	FUNCTION_BLOCK FB 397
	TITLE =G297M FAN KILN 2
	//COPYRIGHT:    (C) 2009  BUHLER AG, CH-9240 UZWIL, SWITZERLAND
	//
	//PRODUCT:      WinCoS_BIW01_09
	//
	//TITLE:        FAN KILN 2
	//                Machine group control
	//                Maschinengruppensteuerung
	//
	//--------------------------------------------------------------------------------
	//
	//IDENT:        AUTHOR:             DEPT:                              DATE:
	//
	//P01_FB397.1.0 K.Renz              CSB41                              20.Mai.2010
	//             1st Release
	//
	//--------------------------------------------------------------------------------
	//
	//PURPOSE:
	//
	//MANUAL :
	//
	//RESTRICTIONS:
	//
	//--------------------------------------------------------------------------------
	AUTHOR  : KR
	FAMILY  : USW
	VERSION : 9.9


	VAR
	  Gr       : FB10;	//Standard interface to group
	  InOutValue1    : DINT; //Data for user
	  InOutValue2    : DINT; //Data for user
	  OutWayConflict : BOOL;	//Data for user
	  OutSelectionOk : BOOL;	//Data for user
	  CmdNewValue : BOOL;	//Data for user
	  CmdNewJob   : BOOL;	//Data for user
	  OutCodeOK   : BOOL;	//Data for user
	  InEndOfJob  : BOOL ;	//Data for user
	  staWayOk      : BOOL ;	//Data for user
	  EdgeStartRelease : BOOL ;	//Data for user
	  USW8  : BOOL;	//Data for user
	  USW9 : BOOL;	//Data for user
	  USW10: BOOL;	//Data for user
	  USW11: BOOL;	//Data for user
	  USW12: BOOL;	//Data for user
	  USW13: BOOL;	//Data for user
	  USW14: BOOL;	//Data for user
	  USW15: BOOL;	//Data for user
	     #A_3225_KCU04AI1 : FB19;   // AnaInp
	     #A_3225_KCU04AI2 : FB19;   // AnaInp
	     #A_3225_BTE05 : FB19;   // AnaInp
	     #A_3225_BTE06 : FB19;   // AnaInp
	     #A_3225_TSC01 : FB14;   // DigInpCont
	     #A_3225_MXZ01MA : FB1032;   // Motor+6DI
	     #A_3225_TSC01_AC : FB19;   // AnaInp
	     #A_3225_TSC01_AF : FB19;   // AnaInp
	     #A_3225_TSC01_AP : FB19;   // AnaInp
	     #A_3225_TSC01_AT : FB19;   // AnaInp
	     #A_3225_TSC01_COM : FB1812;   // FU_Siemens
	     #A_3226_KCU04AI1 : FB19;   // AnaInp
	     #A_3226_KCU04AI2 : FB19;   // AnaInp
	     #A_3226_BTE05 : FB19;   // AnaInp
	     #A_3226_BTE06 : FB19;   // AnaInp
	     #A_3226_MXZ01MA : FB1033;   // Motor+6DI
	     #A_3226_TSC01_AC : FB19;   // AnaInp
	     #A_3226_TSC01_AF : FB19;   // AnaInp
	     #A_3226_TSC01_AP : FB19;   // AnaInp
	     #A_3226_TSC01_AT : FB19;   // AnaInp
	     #A_3226_TSC01_COM : FB1812;   // FU_Siemens
	     #A_3226_TSC01 : FB14;   // DigInpCont
	     #A_3225_MXZ02MA : FB1066;   // Motor+6DI
	     #A_3226_MXZ02MA : FB1067;   // Motor+6DI
	END_VAR
	VAR_TEMP
	   tmpEnable		: BOOL;
	   tmpFlag  		: BOOL;
	   tmpCmdNext		: BOOL;
	   tmpLocal  		: BOOL;
	   tmpAspOk  		: BOOL;
	   tmpHWStop 		: BOOL;
	   tmpInstanzDBNo       : INT ;
	END_VAR
	BEGIN
	NETWORK
	TITLE =
	NETWORK
	TITLE =Read command from group control
	//Parameter
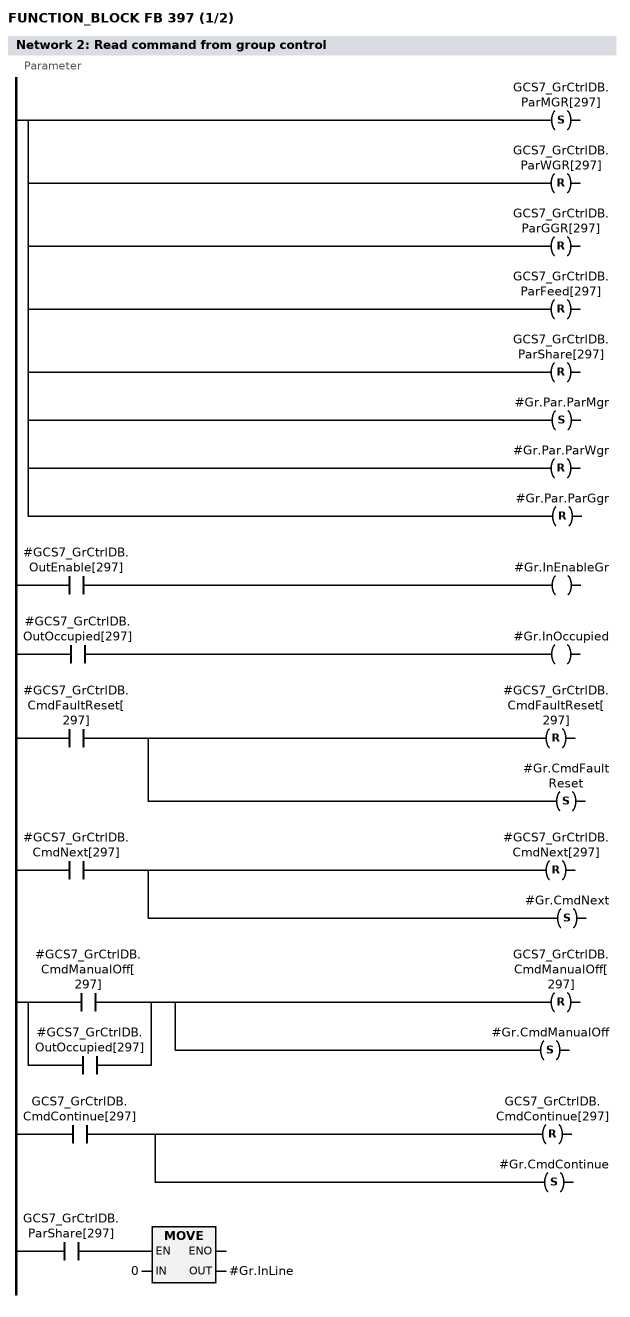
	      SET;
	      S   GCS7_GrCtrlDB.ParMGR[297];
	      R   GCS7_GrCtrlDB.ParWGR[297];
	      R   GCS7_GrCtrlDB.ParGGR[297];
	      R   GCS7_GrCtrlDB.ParFeed[297];
	      R   GCS7_GrCtrlDB.ParShare[297];
	      S   #Gr.Par.ParMgr;
	      R   #Gr.Par.ParWgr;
	      R   #Gr.Par.ParGgr;
	//Command
	      U   #GCS7_GrCtrlDB.OutEnable[297];
	      =   #Gr.InEnableGr;
	      U   #GCS7_GrCtrlDB.OutOccupied[297];
	      =   #Gr.InOccupied;
	      U   #GCS7_GrCtrlDB.CmdFaultReset[297];
	      R   #GCS7_GrCtrlDB.CmdFaultReset[297];
	      S   #Gr.CmdFaultReset;
	      U  #GCS7_GrCtrlDB.CmdNext[297];
	      R   #GCS7_GrCtrlDB.CmdNext[297];
	      S   #Gr.CmdNext;
	      U   #GCS7_GrCtrlDB.CmdManualOff[297];
	      O   #GCS7_GrCtrlDB.OutOccupied[297];
	      R   GCS7_GrCtrlDB.CmdManualOff[297];
	      S   #Gr.CmdManualOff;
	      U  GCS7_GrCtrlDB.CmdContinue[297];
	      R   GCS7_GrCtrlDB.CmdContinue[297];
	      S   #Gr.CmdContinue;
	//Init Line Number
	      U   GCS7_GrCtrlDB.ParShare[297];
	      SPBN WE00;
	      L     0;
	      T     #Gr.InLine;
	WE00: NOP   0;
	NETWORK
	TITLE =Call Methode Control
	// 1. Handle Interface PCControl
	// 2. Prepare mode --> ModePassive,ModeActive,ModeIdling
	// 3. Reset global flags of the group
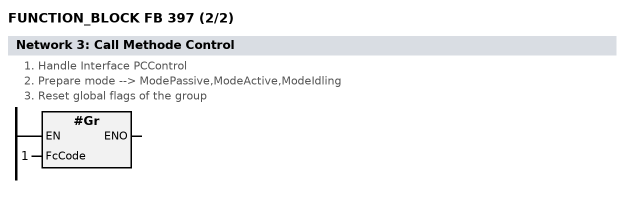
	      CALL #Gr (
	           FcCode                   := 1);
	NETWORK
	TITLE =Restart Idling Time
		L  #Gr.Par.ParIdling;
		L  2;
		>=I;
		SPB IdTm;
		T  #Gr.Par.ParIdling;
	IdTm:   NOP 0;
	      CLR;
	      S    #Gr.CmdRestartIdling;
	NETWORK
	TITLE =Prepare global flags
	NETWORK
	TITLE =Set Pattern (Target position)
	NETWORK
	TITLE =Interlocking WayOk
	//
	NETWORK
	TITLE =Interlocking Autostart
		CLR;
		R   #Gr.OutAutostart;
	NETWORK
	TITLE =Interlocking Enable
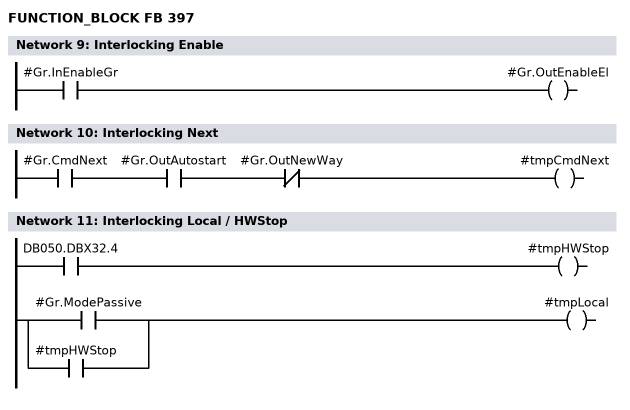
	      U     #Gr.InEnableGr;
	      =     #Gr.OutEnableEl;

	NETWORK
	TITLE =Interlocking Next
	      U     #Gr.CmdNext;
	      U     #Gr.OutAutostart;
	      UN    #Gr.OutNewWay;
	      =    #tmpCmdNext;

	NETWORK
	TITLE =Interlocking Local / HWStop
	      U    DB050.DBX32.4;
	      =    #tmpHWStop;

	      U    #Gr.ModePassive;
	      O    #tmpHWStop;
	      =    #tmpLocal;

	NETWORK
	TITLE =Interlocking Start Warning
	      NOP 0;
	//- Restart after fault --
	      U     #Gr.CmdFaultReset;
	      U     #Gr.VarFault;
	      S       "SYS_StartWarningDB".Area[11].CmdResetStartWarning;
	//- Run Timer --
	      AUF "G297M";
	      CALL  FB100 , DB100(
	       InModeHigher :=FALSE,
	       InArea     :=11,
	       InEnable   :=#Gr.OutEnableEl,
	       InLocal    :=#tmpLocal,
	       InStarted  :=#Gr.VarStarted,
	       InCmdNext  :=#tmpCmdNext,
	       OutCmdNext :=#tmpCmdNext,
	       OutStartwarning:=#Gr.VarStartWarning);
	//- Store Startwarning done  --
	//- Reset Autostart --
	      U     "SYS_StartWarningDB".TmpArea.OutStartReleaseRunningL;
	      FN    #EdgeStartRelease;
	      U     #Gr.VarFault;
	      R     #Gr.OutAutostart;
	NETWORK
	TITLE ==A-3225-KCU04AI1 : VIBRATION MONITOR FAN 1 CHANNEL 1
	NOP 0;
	//-InLocal---
	      U     #tmpLocal;
	      =     #A_3225_KCU04AI1.InLocal;
	//
	//-Monitoring---
	      CLR;
	      =     #A_3225_KCU04AI1.InMonLL;
	      CLR;
	      =     #A_3225_KCU04AI1.InMonL;
	      CLR;
	      =     #A_3225_KCU04AI1.InMonMid;
	      CLR;
	      =     #A_3225_KCU04AI1.InMonH;
	      SET;
	      =     #A_3225_KCU04AI1.InMonHH;
	//
	//-Read inputs---
	      L     PEW1054;
	      T     #A_3225_KCU04AI1.InpValue;
	      U   DB050.DBX32.4;
	      =     #A_3225_KCU04AI1.InHWStop;
	       U     PLC_DPInfo.Master[1].SlavesError[102];
	       =       #A_3225_KCU04AI1.InDPFault;
	//
	//-Set Parameters---
	//
	//-Call object control---
	      CALL  #A_3225_KCU04AI1;
	//
	//-Write outputs---
	NETWORK
	TITLE ==A-3225-KCU04AI2 : VIBRATION MONITOR FAN 1 CHANNEL 2
	NOP 0;
	//-InLocal---
	      U     #tmpLocal;
	      =     #A_3225_KCU04AI2.InLocal;
	//
	//-Monitoring---
	      CLR;
	      =     #A_3225_KCU04AI2.InMonLL;
	      CLR;
	      =     #A_3225_KCU04AI2.InMonL;
	      CLR;
	      =     #A_3225_KCU04AI2.InMonMid;
	      CLR;
	      =     #A_3225_KCU04AI2.InMonH;
	      SET;
	      =     #A_3225_KCU04AI2.InMonHH;
	//
	//-Read inputs---
	      L     PEW1052;
	      T     #A_3225_KCU04AI2.InpValue;
	      U   DB050.DBX32.4;
	      =     #A_3225_KCU04AI2.InHWStop;
	       U     PLC_DPInfo.Master[1].SlavesError[102];
	       =       #A_3225_KCU04AI2.InDPFault;
	//
	//-Set Parameters---
	//
	//-Call object control---
	      CALL  #A_3225_KCU04AI2;
	//
	//-Write outputs---
	NETWORK
	TITLE ==A-3225-BTE05 : TEMPERATURE BEARING TEMPERATUR SENSOR
	NOP 0;
	//-InLocal---
	      U     #tmpLocal;
	      =     #A_3225_BTE05.InLocal;
	//
	//-Monitoring---
	      CLR;
	      =     #A_3225_BTE05.InMonLL;
	      CLR;
	      =     #A_3225_BTE05.InMonL;
	      CLR;
	      =     #A_3225_BTE05.InMonMid;
	      CLR;
	      =     #A_3225_BTE05.InMonH;
	      SET;
	      =     #A_3225_BTE05.InMonHH;
	//
	//-Read inputs---
	      L     PEW1028;
	      T     #A_3225_BTE05.InpValue;
	      U   DB050.DBX32.4;
	      =     #A_3225_BTE05.InHWStop;
	       U     PLC_DPInfo.Master[1].SlavesError[102];
	       =       #A_3225_BTE05.InDPFault;
	//
	//-Set Parameters---
	//
	//-Call object control---
	      CALL  #A_3225_BTE05;
	//
	//-Write outputs---
	NETWORK
	TITLE ==A-3225-BTE06 : TEMPERATURE BEARING TEMPERATUR SENSOR
	NOP 0;
	//-InLocal---
	      U     #tmpLocal;
	      =     #A_3225_BTE06.InLocal;
	//
	//-Monitoring---
	      CLR;
	      =     #A_3225_BTE06.InMonLL;
	      CLR;
	      =     #A_3225_BTE06.InMonL;
	      CLR;
	      =     #A_3225_BTE06.InMonMid;
	      CLR;
	      =     #A_3225_BTE06.InMonH;
	      SET;
	      =     #A_3225_BTE06.InMonHH;
	//
	//-Read inputs---
	      L     PEW1030;
	      T     #A_3225_BTE06.InpValue;
	      U   DB050.DBX32.4;
	      =     #A_3225_BTE06.InHWStop;
	       U     PLC_DPInfo.Master[1].SlavesError[102];
	       =       #A_3225_BTE06.InDPFault;
	//
	//-Set Parameters---
	//
	//-Call object control---
	      CALL  #A_3225_BTE06;
	//
	//-Write outputs---
	NETWORK
	TITLE ==A-3225-MXZ02MA : GETRIEBEÖLPUMPE FAN 1
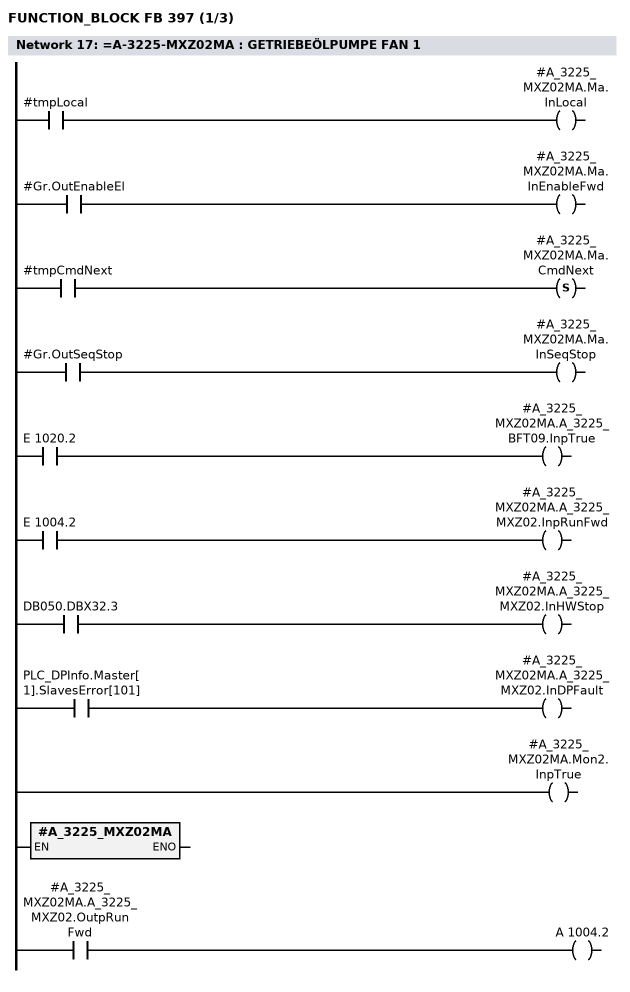
	NOP 0;
	//-InLocal---
	      U     #tmpLocal;
	      =     #A_3225_MXZ02MA.Ma.InLocal;
	//
	//-Interlocking---

	      U     #Gr.OutEnableEl;
	      =     #A_3225_MXZ02MA.Ma.InEnableFwd;
	//
	      U    #tmpCmdNext;
	      S     #A_3225_MXZ02MA.Ma.CmdNext;
	//
	      U     #Gr.OutSeqStop;
	      =     #A_3225_MXZ02MA.Ma.InSeqStop;
	//
	//=Values and commands of elements===
	//-=A-3225-BFT09---
	//      CLR
	//      S     #A_3225_MXZ02MA.A_3225_BFT09.CmdRunTimeOutTime
	//
	//-Read inputs of elements---
	      U     E 1020.2;
	      =     #A_3225_MXZ02MA.A_3225_BFT09.InpTrue;
	      U     E 1004.2;
	      =     #A_3225_MXZ02MA.A_3225_MXZ02.InpRunFwd;
	      U   DB050.DBX32.3;
	      =     #A_3225_MXZ02MA.A_3225_MXZ02.InHWStop;
	       U     PLC_DPInfo.Master[1].SlavesError[101];
	       =       #A_3225_MXZ02MA.A_3225_MXZ02.InDPFault;
	      SET;
	      =     #A_3225_MXZ02MA.Mon2.InpTrue;
	//
	//-Set Parameters---
	//
	//-Call object control---
	      CALL  #A_3225_MXZ02MA;
	//
	//-Write outputs---
	      U     #A_3225_MXZ02MA.A_3225_MXZ02.OutpRunFwd;
	      =     A 1004.2;
	NETWORK
	TITLE ==A-3225-MXZ01MA : FAN 1
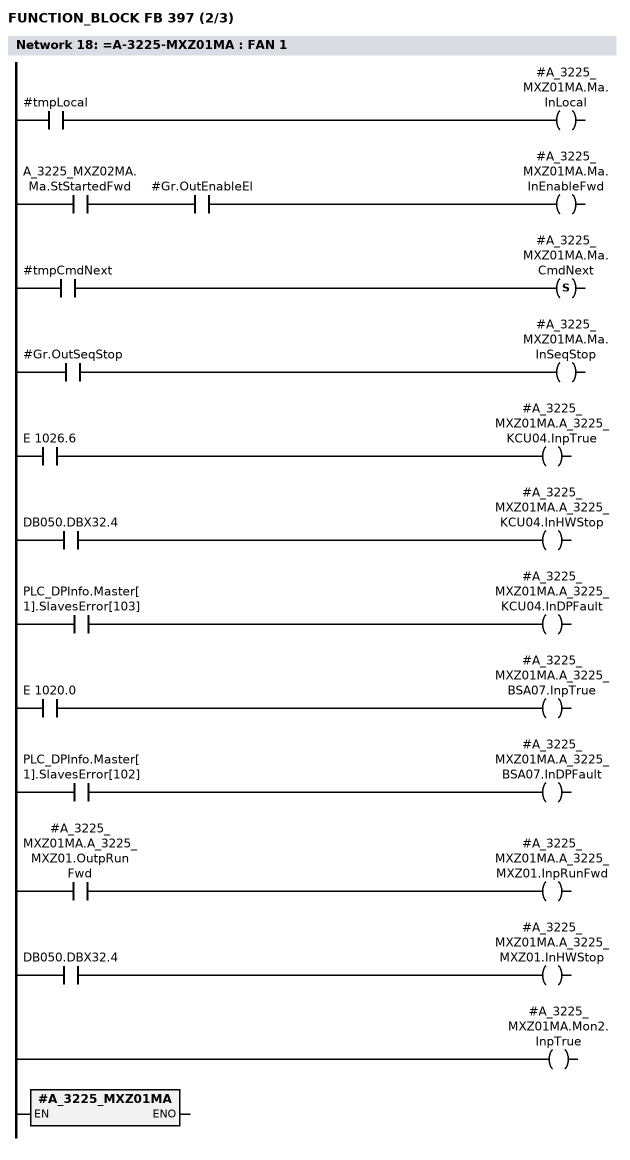
	NOP 0;
	//-InLocal---
	      U     #tmpLocal;
	      =     #A_3225_MXZ01MA.Ma.InLocal;
	//
	//-Interlocking---
	      U A_3225_MXZ02MA.Ma.StStartedFwd;
	      U     #Gr.OutEnableEl;
	      =     #A_3225_MXZ01MA.Ma.InEnableFwd;
	//
	      U    #tmpCmdNext;
	      S     #A_3225_MXZ01MA.Ma.CmdNext;
	//
	      U     #Gr.OutSeqStop;
	      =     #A_3225_MXZ01MA.Ma.InSeqStop;
	//
	//=Values and commands of elements===
	//-=A-3225-KCU04---
	//      CLR
	//      S     #A_3225_MXZ01MA.A_3225_KCU04.CmdRunTimeOutTime
	//-=A-3225-BSA07---
	//      CLR
	//      S     #A_3225_MXZ01MA.A_3225_BSA07.CmdRunTimeOutTime
	//
	//-Read inputs of elements---
	      U     E 1026.6;
	      =     #A_3225_MXZ01MA.A_3225_KCU04.InpTrue;
	      U   DB050.DBX32.4;
	      =     #A_3225_MXZ01MA.A_3225_KCU04.InHWStop;
	       U     PLC_DPInfo.Master[1].SlavesError[103];
	       =       #A_3225_MXZ01MA.A_3225_KCU04.InDPFault;
	      U     E 1020.0;
	      =     #A_3225_MXZ01MA.A_3225_BSA07.InpTrue;
	       U     PLC_DPInfo.Master[1].SlavesError[102];
	       =       #A_3225_MXZ01MA.A_3225_BSA07.InDPFault;
	      U     #A_3225_MXZ01MA.A_3225_MXZ01.OutpRunFwd;
	      =     #A_3225_MXZ01MA.A_3225_MXZ01.InpRunFwd;
	      U   DB050.DBX32.4;
	      =     #A_3225_MXZ01MA.A_3225_MXZ01.InHWStop;
	      SET;
	      =     #A_3225_MXZ01MA.Mon2.InpTrue;
	//
	//-Set Parameters---
	//
	//-Call object control---
	      CALL  #A_3225_MXZ01MA;
	//
	//-Write outputs---
	NETWORK
	TITLE ==A-3225-TSC01_COM : FAN 1 FU KOMMUNIKATION
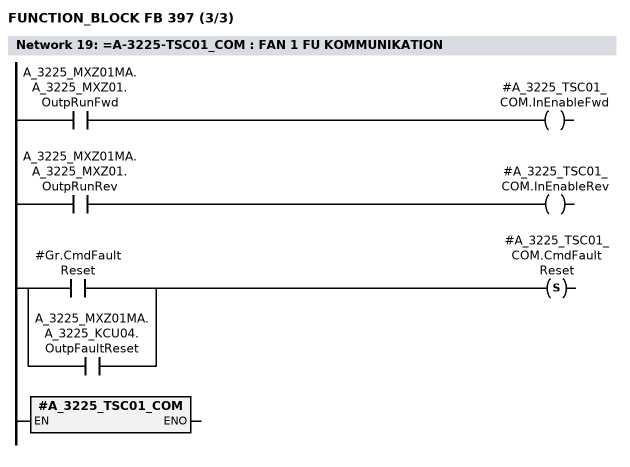
	NOP 0;
	     U   A_3225_MXZ01MA.A_3225_MXZ01.OutpRunFwd;
	      =     #A_3225_TSC01_COM.InEnableFwd;
	     U    A_3225_MXZ01MA.A_3225_MXZ01.OutpRunRev;
	      =     #A_3225_TSC01_COM.InEnableRev;
	     U     #Gr.CmdFaultReset;
	     O    A_3225_MXZ01MA.A_3225_KCU04.OutpFaultReset;
	      S     #A_3225_TSC01_COM.CmdFaultReset;
	//
	//
	//-Read inputs---
	//
	//-Set Parameters---
	//
	//-Call object control---
	      CALL  #A_3225_TSC01_COM;
	//
	//-Write outputs---
	NETWORK
	TITLE ==A-3225-TSC01_AC : ACT. CURRENT FAN 1 FU
	NOP 0;
	//-InLocal---
	      U     #tmpLocal;
	      =     #A_3225_TSC01_AC.InLocal;
	//
	//-Monitoring---
	      CLR;
	      =     #A_3225_TSC01_AC.InMonLL;
	      CLR;
	      =     #A_3225_TSC01_AC.InMonL;
	      CLR;
	      =     #A_3225_TSC01_AC.InMonMid;
	      CLR;
	      =     #A_3225_TSC01_AC.InMonH;
	      CLR;
	      =     #A_3225_TSC01_AC.InMonHH;
	//
	//-Read inputs---
	      L     A_3225_TSC01_COM.Output.SetpointValue01;
	      ITD;
	      DTR;
	      ABS;
	      RND;
	      T     #A_3225_TSC01_AC.InpValue;
	      U   DB050.DBX32.4;
	      =     #A_3225_TSC01_AC.InHWStop;
	//
	//-Set Parameters---
	//
	//-Call object control---
	      CALL  #A_3225_TSC01_AC;
	//
	//-Write outputs---
	NETWORK
	TITLE ==A-3225-TSC01_AF : ACT. FREQUENCY FAN 1 FU
	NOP 0;
	//-InLocal---
	      U     #tmpLocal;
	      =     #A_3225_TSC01_AF.InLocal;
	//
	//-Monitoring---
	      CLR;
	      =     #A_3225_TSC01_AF.InMonLL;
	      CLR;
	      =     #A_3225_TSC01_AF.InMonL;
	      CLR;
	      =     #A_3225_TSC01_AF.InMonMid;
	      CLR;
	      =     #A_3225_TSC01_AF.InMonH;
	      CLR;
	      =     #A_3225_TSC01_AF.InMonHH;
	//
	//-Read inputs---
	      L     A_3225_TSC01_COM.Output.SetpointValue01;
	      ITD;
	      DTR;
	      ABS;
	      RND;
	      T     #A_3225_TSC01_AF.InpValue;
	      U   DB050.DBX32.4;
	      =     #A_3225_TSC01_AF.InHWStop;
	//
	//-Set Parameters---
	//
	//-Call object control---
	      CALL  #A_3225_TSC01_AF;
	//
	//-Write outputs---
	NETWORK
	TITLE ==A-3225-TSC01_AP : ACT. POWER FAN 1 FU
	NOP 0;
	//-InLocal---
	      U     #tmpLocal;
	      =     #A_3225_TSC01_AP.InLocal;
	//
	//-Monitoring---
	      CLR;
	      =     #A_3225_TSC01_AP.InMonLL;
	      CLR;
	      =     #A_3225_TSC01_AP.InMonL;
	      CLR;
	      =     #A_3225_TSC01_AP.InMonMid;
	      CLR;
	      =     #A_3225_TSC01_AP.InMonH;
	      CLR;
	      =     #A_3225_TSC01_AP.InMonHH;
	//
	//-Read inputs---
	      L     A_3225_TSC01_COM.Output.SetpointValue01;
	      ITD;
	      DTR;
	      ABS;
	      RND;
	      T     #A_3225_TSC01_AP.InpValue;
	      U   DB050.DBX32.4;
	      =     #A_3225_TSC01_AP.InHWStop;
	//
	//-Set Parameters---
	//
	//-Call object control---
	      CALL  #A_3225_TSC01_AP;
	//
	//-Write outputs---
	NETWORK
	TITLE ==A-3225-TSC01_AT : ACT. TORQUE FAN 1 FU
	NOP 0;
	//-InLocal---
	      U     #tmpLocal;
	      =     #A_3225_TSC01_AT.InLocal;
	//
	//-Monitoring---
	      CLR;
	      =     #A_3225_TSC01_AT.InMonLL;
	      CLR;
	      =     #A_3225_TSC01_AT.InMonL;
	      CLR;
	      =     #A_3225_TSC01_AT.InMonMid;
	      CLR;
	      =     #A_3225_TSC01_AT.InMonH;
	      CLR;
	      =     #A_3225_TSC01_AT.InMonHH;
	//
	//-Read inputs---
	      L     A_3225_TSC01_COM.Output.SetpointValue01;
	      ITD;
	      DTR;
	      ABS;
	      RND;
	      T     #A_3225_TSC01_AT.InpValue;
	      U   DB050.DBX32.4;
	      =     #A_3225_TSC01_AT.InHWStop;
	//
	//-Set Parameters---
	//
	//-Call object control---
	      CALL  #A_3225_TSC01_AT;
	//
	//-Write outputs---
	NETWORK
	TITLE ==A-3226-KCU04AI1 : VIBRATION MONITOR FAN 2 CHANNEL 1
	NOP 0;
	//-InLocal---
	      U     #tmpLocal;
	      =     #A_3226_KCU04AI1.InLocal;
	//
	//-Monitoring---
	      CLR;
	      =     #A_3226_KCU04AI1.InMonLL;
	      CLR;
	      =     #A_3226_KCU04AI1.InMonL;
	      CLR;
	      =     #A_3226_KCU04AI1.InMonMid;
	      CLR;
	      =     #A_3226_KCU04AI1.InMonH;
	      SET;
	      =     #A_3226_KCU04AI1.InMonHH;
	//
	//-Read inputs---
	      L     PEW1058;
	      T     #A_3226_KCU04AI1.InpValue;
	      U   DB050.DBX32.4;
	      =     #A_3226_KCU04AI1.InHWStop;
	       U     PLC_DPInfo.Master[1].SlavesError[102];
	       =       #A_3226_KCU04AI1.InDPFault;
	//
	//-Set Parameters---
	//
	//-Call object control---
	      CALL  #A_3226_KCU04AI1;
	//
	//-Write outputs---
	NETWORK
	TITLE ==A-3226-KCU04AI2 : VIBRATION MONITOR FAN 2 CHANNEL 2
	NOP 0;
	//-InLocal---
	      U     #tmpLocal;
	      =     #A_3226_KCU04AI2.InLocal;
	//
	//-Monitoring---
	      CLR;
	      =     #A_3226_KCU04AI2.InMonLL;
	      CLR;
	      =     #A_3226_KCU04AI2.InMonL;
	      CLR;
	      =     #A_3226_KCU04AI2.InMonMid;
	      CLR;
	      =     #A_3226_KCU04AI2.InMonH;
	      SET;
	      =     #A_3226_KCU04AI2.InMonHH;
	//
	//-Read inputs---
	      L     PEW1056;
	      T     #A_3226_KCU04AI2.InpValue;
	      U   DB050.DBX32.4;
	      =     #A_3226_KCU04AI2.InHWStop;
	       U     PLC_DPInfo.Master[1].SlavesError[102];
	       =       #A_3226_KCU04AI2.InDPFault;
	//
	//-Set Parameters---
	//
	//-Call object control---
	      CALL  #A_3226_KCU04AI2;
	//
	//-Write outputs---
	NETWORK
	TITLE ==A-3226-BTE05 : TEMPERATURE BEARING TEMPERATUR SENSOR
	NOP 0;
	//-InLocal---
	      U     #tmpLocal;
	      =     #A_3226_BTE05.InLocal;
	//
	//-Monitoring---
	      CLR;
	      =     #A_3226_BTE05.InMonLL;
	      CLR;
	      =     #A_3226_BTE05.InMonL;
	      CLR;
	      =     #A_3226_BTE05.InMonMid;
	      CLR;
	      =     #A_3226_BTE05.InMonH;
	      SET;
	      =     #A_3226_BTE05.InMonHH;
	//
	//-Read inputs---
	      L     PEW1032;
	      T     #A_3226_BTE05.InpValue;
	      U   DB050.DBX32.4;
	      =     #A_3226_BTE05.InHWStop;
	       U     PLC_DPInfo.Master[1].SlavesError[102];
	       =       #A_3226_BTE05.InDPFault;
	//
	//-Set Parameters---
	//
	//-Call object control---
	      CALL  #A_3226_BTE05;
	//
	//-Write outputs---
	NETWORK
	TITLE ==A-3226-BTE06 : TEMPERATURE BEARING TEMPERATUR SENSOR
	NOP 0;
	//-InLocal---
	      U     #tmpLocal;
	      =     #A_3226_BTE06.InLocal;
	//
	//-Monitoring---
	      CLR;
	      =     #A_3226_BTE06.InMonLL;
	      CLR;
	      =     #A_3226_BTE06.InMonL;
	      CLR;
	      =     #A_3226_BTE06.InMonMid;
	      CLR;
	      =     #A_3226_BTE06.InMonH;
	      SET;
	      =     #A_3226_BTE06.InMonHH;
	//
	//-Read inputs---
	      L     PEW1034;
	      T     #A_3226_BTE06.InpValue;
	      U   DB050.DBX32.4;
	      =     #A_3226_BTE06.InHWStop;
	       U     PLC_DPInfo.Master[1].SlavesError[102];
	       =       #A_3226_BTE06.InDPFault;
	//
	//-Set Parameters---
	//
	//-Call object control---
	      CALL  #A_3226_BTE06;
	//
	//-Write outputs---
	NETWORK
	TITLE ==A-3226-MXZ02MA : GETRIEBEÖLPUMPE FAN 2
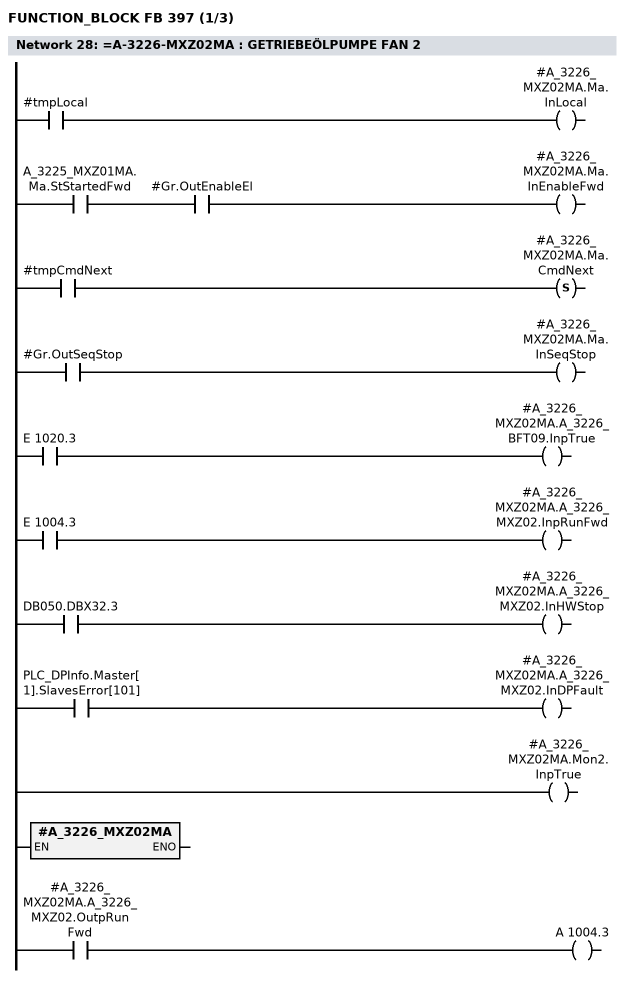
	NOP 0;
	//-InLocal---
	      U     #tmpLocal;
	      =     #A_3226_MXZ02MA.Ma.InLocal;
	//
	//-Interlocking---
	      U A_3225_MXZ01MA.Ma.StStartedFwd;
	      U     #Gr.OutEnableEl;
	      =     #A_3226_MXZ02MA.Ma.InEnableFwd;
	//
	      U    #tmpCmdNext;
	      S     #A_3226_MXZ02MA.Ma.CmdNext;
	//
	      U     #Gr.OutSeqStop;
	      =     #A_3226_MXZ02MA.Ma.InSeqStop;
	//
	//=Values and commands of elements===
	//-=A-3226-BFT09---
	//      CLR
	//      S     #A_3226_MXZ02MA.A_3226_BFT09.CmdRunTimeOutTime
	//
	//-Read inputs of elements---
	      U     E 1020.3;
	      =     #A_3226_MXZ02MA.A_3226_BFT09.InpTrue;
	      U     E 1004.3;
	      =     #A_3226_MXZ02MA.A_3226_MXZ02.InpRunFwd;
	      U   DB050.DBX32.3;
	      =     #A_3226_MXZ02MA.A_3226_MXZ02.InHWStop;
	       U     PLC_DPInfo.Master[1].SlavesError[101];
	       =       #A_3226_MXZ02MA.A_3226_MXZ02.InDPFault;
	      SET;
	      =     #A_3226_MXZ02MA.Mon2.InpTrue;
	//
	//-Set Parameters---
	//
	//-Call object control---
	      CALL  #A_3226_MXZ02MA;
	//
	//-Write outputs---
	      U     #A_3226_MXZ02MA.A_3226_MXZ02.OutpRunFwd;
	      =     A 1004.3;
	NETWORK
	TITLE ==A-3226-MXZ01MA : FAN 2
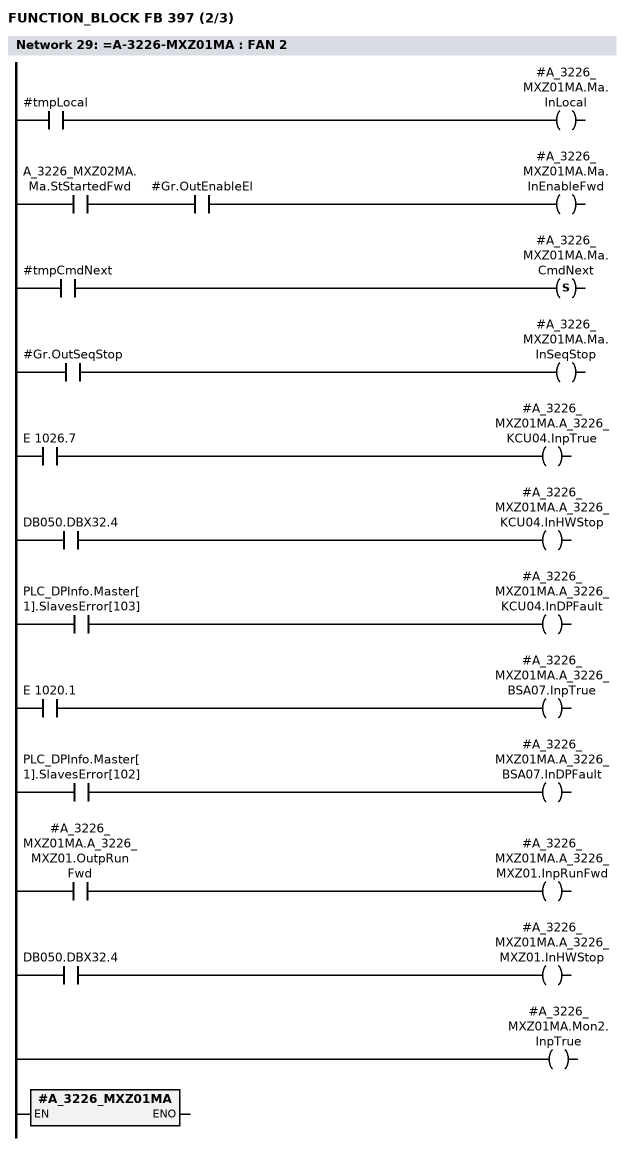
	NOP 0;
	//-InLocal---
	      U     #tmpLocal;
	      =     #A_3226_MXZ01MA.Ma.InLocal;
	//
	//-Interlocking---
	      U A_3226_MXZ02MA.Ma.StStartedFwd;
	      U     #Gr.OutEnableEl;
	      =     #A_3226_MXZ01MA.Ma.InEnableFwd;
	//
	      U    #tmpCmdNext;
	      S     #A_3226_MXZ01MA.Ma.CmdNext;
	//
	      U     #Gr.OutSeqStop;
	      =     #A_3226_MXZ01MA.Ma.InSeqStop;
	//
	//=Values and commands of elements===
	//-=A-3226-KCU04---
	//      CLR
	//      S     #A_3226_MXZ01MA.A_3226_KCU04.CmdRunTimeOutTime
	//-=A-3226-BSA07---
	//      CLR
	//      S     #A_3226_MXZ01MA.A_3226_BSA07.CmdRunTimeOutTime
	//
	//-Read inputs of elements---
	      U     E 1026.7;
	      =     #A_3226_MXZ01MA.A_3226_KCU04.InpTrue;
	      U   DB050.DBX32.4;
	      =     #A_3226_MXZ01MA.A_3226_KCU04.InHWStop;
	       U     PLC_DPInfo.Master[1].SlavesError[103];
	       =       #A_3226_MXZ01MA.A_3226_KCU04.InDPFault;
	      U     E 1020.1;
	      =     #A_3226_MXZ01MA.A_3226_BSA07.InpTrue;
	       U     PLC_DPInfo.Master[1].SlavesError[102];
	       =       #A_3226_MXZ01MA.A_3226_BSA07.InDPFault;
	      U     #A_3226_MXZ01MA.A_3226_MXZ01.OutpRunFwd;
	      =     #A_3226_MXZ01MA.A_3226_MXZ01.InpRunFwd;
	      U   DB050.DBX32.4;
	      =     #A_3226_MXZ01MA.A_3226_MXZ01.InHWStop;
	      SET;
	      =     #A_3226_MXZ01MA.Mon2.InpTrue;
	//
	//-Set Parameters---
	//
	//-Call object control---
	      CALL  #A_3226_MXZ01MA;
	//
	//-Write outputs---
	NETWORK
	TITLE ==A-3226-TSC01_COM : FAN 2 FU KOMMUNIKATION
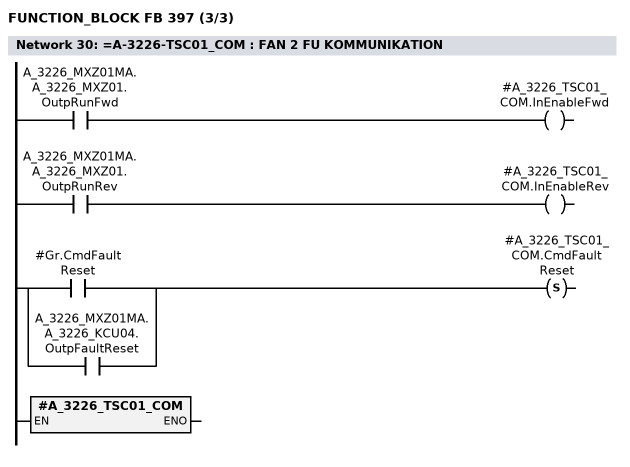
	NOP 0;
	     U   A_3226_MXZ01MA.A_3226_MXZ01.OutpRunFwd;
	      =     #A_3226_TSC01_COM.InEnableFwd;
	     U    A_3226_MXZ01MA.A_3226_MXZ01.OutpRunRev;
	      =     #A_3226_TSC01_COM.InEnableRev;
	     U     #Gr.CmdFaultReset;
	     O    A_3226_MXZ01MA.A_3226_KCU04.OutpFaultReset;
	      S     #A_3226_TSC01_COM.CmdFaultReset;
	//
	//
	//-Read inputs---
	//
	//-Set Parameters---
	//
	//-Call object control---
	      CALL  #A_3226_TSC01_COM;
	//
	//-Write outputs---
	NETWORK
	TITLE ==A-3226-TSC01_AC : ACT. CURRENT FAN 2 FU
	NOP 0;
	//-InLocal---
	      U     #tmpLocal;
	      =     #A_3226_TSC01_AC.InLocal;
	//
	//-Monitoring---
	      CLR;
	      =     #A_3226_TSC01_AC.InMonLL;
	      CLR;
	      =     #A_3226_TSC01_AC.InMonL;
	      CLR;
	      =     #A_3226_TSC01_AC.InMonMid;
	      CLR;
	      =     #A_3226_TSC01_AC.InMonH;
	      CLR;
	      =     #A_3226_TSC01_AC.InMonHH;
	//
	//-Read inputs---
	      L     A_3226_TSC01_COM.Output.SetpointValue01;
	      ITD;
	      DTR;
	      ABS;
	      RND;
	      T     #A_3226_TSC01_AC.InpValue;
	      U   DB050.DBX32.4;
	      =     #A_3226_TSC01_AC.InHWStop;
	//
	//-Set Parameters---
	//
	//-Call object control---
	      CALL  #A_3226_TSC01_AC;
	//
	//-Write outputs---
	NETWORK
	TITLE ==A-3226-TSC01_AF : ACT. FREQUENCY FAN 2 FU
	NOP 0;
	//-InLocal---
	      U     #tmpLocal;
	      =     #A_3226_TSC01_AF.InLocal;
	//
	//-Monitoring---
	      CLR;
	      =     #A_3226_TSC01_AF.InMonLL;
	      CLR;
	      =     #A_3226_TSC01_AF.InMonL;
	      CLR;
	      =     #A_3226_TSC01_AF.InMonMid;
	      CLR;
	      =     #A_3226_TSC01_AF.InMonH;
	      CLR;
	      =     #A_3226_TSC01_AF.InMonHH;
	//
	//-Read inputs---
	      L     A_3226_TSC01_COM.Output.SetpointValue01;
	      ITD;
	      DTR;
	      ABS;
	      RND;
	      T     #A_3226_TSC01_AF.InpValue;
	      U   DB050.DBX32.4;
	      =     #A_3226_TSC01_AF.InHWStop;
	//
	//-Set Parameters---
	//
	//-Call object control---
	      CALL  #A_3226_TSC01_AF;
	//
	//-Write outputs---
	NETWORK
	TITLE ==A-3226-TSC01_AP : ACT. POWER FAN 2 FU
	NOP 0;
	//-InLocal---
	      U     #tmpLocal;
	      =     #A_3226_TSC01_AP.InLocal;
	//
	//-Monitoring---
	      CLR;
	      =     #A_3226_TSC01_AP.InMonLL;
	      CLR;
	      =     #A_3226_TSC01_AP.InMonL;
	      CLR;
	      =     #A_3226_TSC01_AP.InMonMid;
	      CLR;
	      =     #A_3226_TSC01_AP.InMonH;
	      CLR;
	      =     #A_3226_TSC01_AP.InMonHH;
	//
	//-Read inputs---
	      L     A_3226_TSC01_COM.Output.SetpointValue01;
	      ITD;
	      DTR;
	      ABS;
	      RND;
	      T     #A_3226_TSC01_AP.InpValue;
	      U   DB050.DBX32.4;
	      =     #A_3226_TSC01_AP.InHWStop;
	//
	//-Set Parameters---
	//
	//-Call object control---
	      CALL  #A_3226_TSC01_AP;
	//
	//-Write outputs---
	NETWORK
	TITLE ==A-3226-TSC01_AT : ACT. TORQUE FAN 2 FU
	NOP 0;
	//-InLocal---
	      U     #tmpLocal;
	      =     #A_3226_TSC01_AT.InLocal;
	//
	//-Monitoring---
	      CLR;
	      =     #A_3226_TSC01_AT.InMonLL;
	      CLR;
	      =     #A_3226_TSC01_AT.InMonL;
	      CLR;
	      =     #A_3226_TSC01_AT.InMonMid;
	      CLR;
	      =     #A_3226_TSC01_AT.InMonH;
	      CLR;
	      =     #A_3226_TSC01_AT.InMonHH;
	//
	//-Read inputs---
	      L     A_3226_TSC01_COM.Output.SetpointValue01;
	      ITD;
	      DTR;
	      ABS;
	      RND;
	      T     #A_3226_TSC01_AT.InpValue;
	      U   DB050.DBX32.4;
	      =     #A_3226_TSC01_AT.InHWStop;
	//
	//-Set Parameters---
	//
	//-Call object control---
	      CALL  #A_3226_TSC01_AT;
	//
	//-Write outputs---
	NETWORK
	TITLE ==A-3225-TSC01 : FAN 1 FU KOMMUNIKATION
	NOP 0;
	//-InLocal---
	      U     #tmpLocal;
	      =     #A_3225_TSC01.InLocal;
	//
	//-Monitoring---
	      CLR;
	      =      #A_3225_TSC01.InMonTrue;
	      CLR;
	      =      #A_3225_TSC01.InMonFalse;
	//
	//-PreAlarm---
	      CLR;
	      =      #A_3225_TSC01.InPreAlarmTrue;
	      CLR;
	      =      #A_3225_TSC01.InPreAlarmFalse;
	//
	//-Additional commands---
	//      CLR
	//      S     #A_3225_TSC01.CmdRunTimeOutTime
	//
	//-Read inputs---
	      U     M 050.0;
	      =     #A_3225_TSC01.InpTrue;
	//
	//-Set Parameters---
	//
	//-Call object control---
	      CALL  #A_3225_TSC01;
	//
	//-Write outputs---
	NETWORK
	TITLE ==A-3226-TSC01 : FAN 2 FU KOMMUNIKATION
	NOP 0;
	//-InLocal---
	      U     #tmpLocal;
	      =     #A_3226_TSC01.InLocal;
	//
	//-Monitoring---
	      CLR;
	      =      #A_3226_TSC01.InMonTrue;
	      CLR;
	      =      #A_3226_TSC01.InMonFalse;
	//
	//-PreAlarm---
	      CLR;
	      =      #A_3226_TSC01.InPreAlarmTrue;
	      CLR;
	      =      #A_3226_TSC01.InPreAlarmFalse;
	//
	//-Additional commands---
	//      CLR
	//      S     #A_3226_TSC01.CmdRunTimeOutTime
	//
	//-Read inputs---
	      U     M 050.0;
	      =     #A_3226_TSC01.InpTrue;
	//
	//-Set Parameters---
	//
	//-Call object control---
	      CALL  #A_3226_TSC01;
	//
	//-Write outputs---
	NETWORK
	TITLE =Test Fault
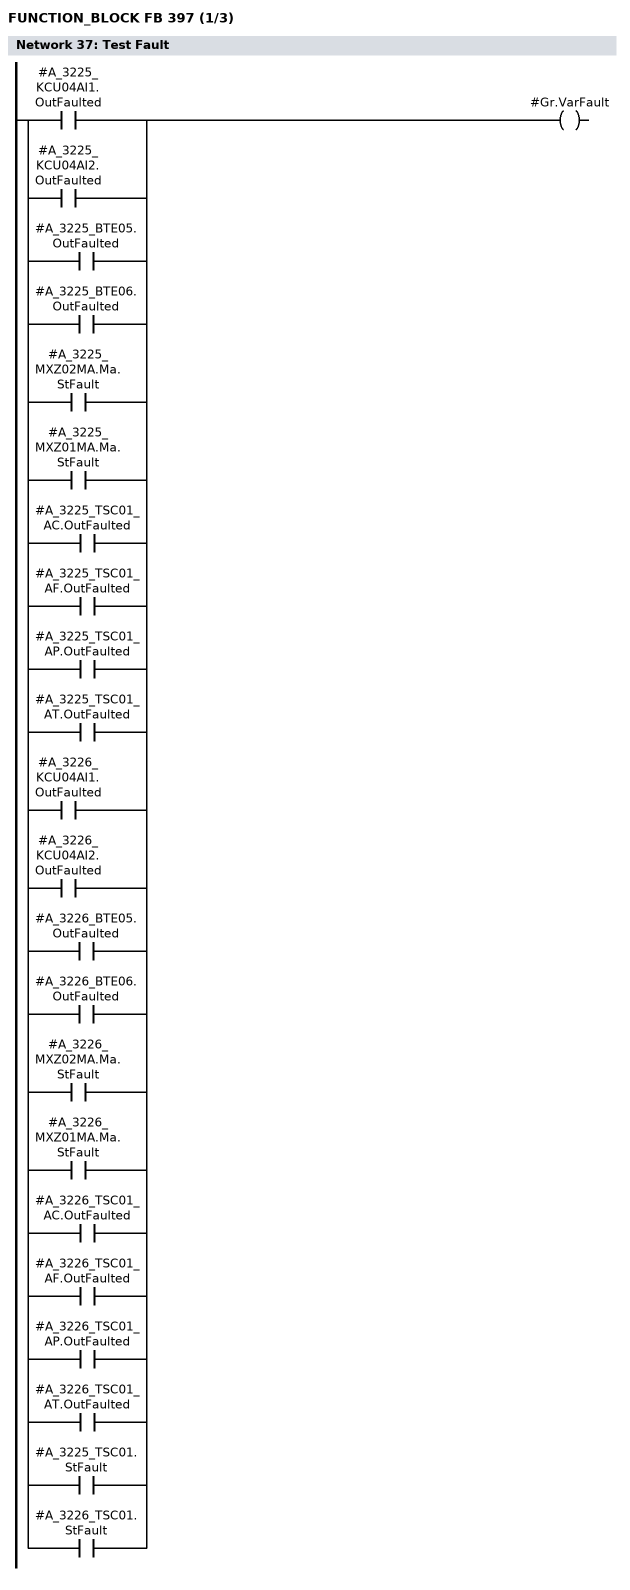
	      U     #A_3225_KCU04AI1.OutFaulted;
	      O     #A_3225_KCU04AI2.OutFaulted;
	      O     #A_3225_BTE05.OutFaulted;
	      O     #A_3225_BTE06.OutFaulted;
	      O     #A_3225_MXZ02MA.Ma.StFault;
	      O     #A_3225_MXZ01MA.Ma.StFault;
	      O     #A_3225_TSC01_AC.OutFaulted;
	      O     #A_3225_TSC01_AF.OutFaulted;
	      O     #A_3225_TSC01_AP.OutFaulted;
	      O     #A_3225_TSC01_AT.OutFaulted;
	      O     #A_3226_KCU04AI1.OutFaulted;
	      O     #A_3226_KCU04AI2.OutFaulted;
	      O     #A_3226_BTE05.OutFaulted;
	      O     #A_3226_BTE06.OutFaulted;
	      O     #A_3226_MXZ02MA.Ma.StFault;
	      O     #A_3226_MXZ01MA.Ma.StFault;
	      O     #A_3226_TSC01_AC.OutFaulted;
	      O     #A_3226_TSC01_AF.OutFaulted;
	      O     #A_3226_TSC01_AP.OutFaulted;
	      O     #A_3226_TSC01_AT.OutFaulted;
	      O     #A_3225_TSC01.StFault;
	      O     #A_3226_TSC01.StFault;
	      =     #Gr.VarFault;
	NETWORK
	TITLE =Test Warning
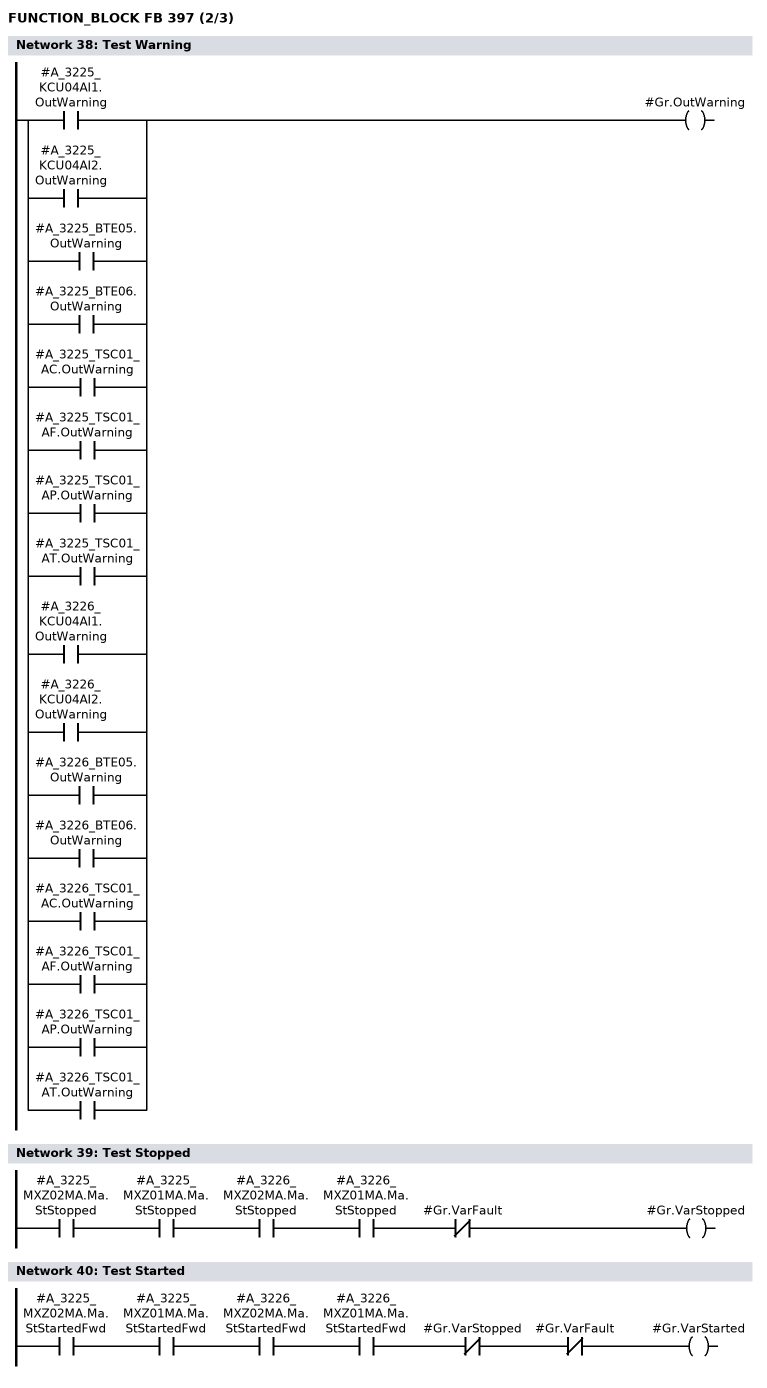
	      U     #A_3225_KCU04AI1.OutWarning;
	      O     #A_3225_KCU04AI2.OutWarning;
	      O     #A_3225_BTE05.OutWarning;
	      O     #A_3225_BTE06.OutWarning;
	      O     #A_3225_TSC01_AC.OutWarning;
	      O     #A_3225_TSC01_AF.OutWarning;
	      O     #A_3225_TSC01_AP.OutWarning;
	      O     #A_3225_TSC01_AT.OutWarning;
	      O     #A_3226_KCU04AI1.OutWarning;
	      O     #A_3226_KCU04AI2.OutWarning;
	      O     #A_3226_BTE05.OutWarning;
	      O     #A_3226_BTE06.OutWarning;
	      O     #A_3226_TSC01_AC.OutWarning;
	      O     #A_3226_TSC01_AF.OutWarning;
	      O     #A_3226_TSC01_AP.OutWarning;
	      O     #A_3226_TSC01_AT.OutWarning;
	      =     #Gr.OutWarning;
	NETWORK
	TITLE =Test Stopped
	      U     #A_3225_MXZ02MA.Ma.StStopped;
	      U     #A_3225_MXZ01MA.Ma.StStopped;
	      U     #A_3226_MXZ02MA.Ma.StStopped;
	      U     #A_3226_MXZ01MA.Ma.StStopped;
	      UN   #Gr.VarFault;
	      =     #Gr.VarStopped;
	NETWORK
	TITLE =Test Started
	      U     #A_3225_MXZ02MA.Ma.StStartedFwd;
	      U     #A_3225_MXZ01MA.Ma.StStartedFwd;
	      U     #A_3226_MXZ02MA.Ma.StStartedFwd;
	      U     #A_3226_MXZ01MA.Ma.StStartedFwd;
	      UN  #Gr.VarStopped;
	      UN  #Gr.VarFault;
	      =     #Gr.VarStarted;
	NETWORK
	TITLE =Enable Previous Group
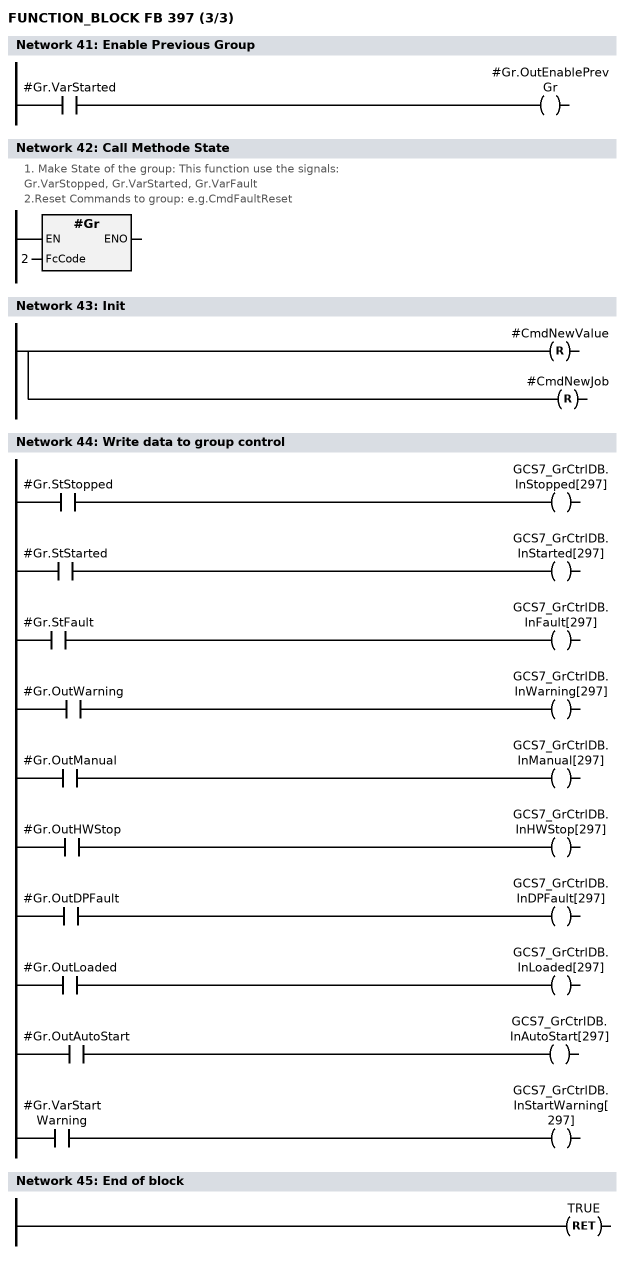
	      U    #Gr.VarStarted;
	      =     #Gr.OutEnablePrevGr;
	NETWORK
	TITLE =Call Methode State
	//1. Make State of the group: This function use the signals:
	//        Gr.VarStopped, Gr.VarStarted, Gr.VarFault
	//2.Reset Commands to group: e.g.CmdFaultReset
	      CALL #Gr (
	           FcCode                   := 2);
	NETWORK
	TITLE =Init
	      SET;
	      R    #CmdNewValue;
	      R    #CmdNewJob;
	NETWORK
	TITLE =Write data to group control
	      U   #Gr.StStopped;
	      =   GCS7_GrCtrlDB.InStopped[297];
	      U   #Gr.StStarted;
	      =   GCS7_GrCtrlDB.InStarted[297];
	      U   #Gr.StFault;
	      =   GCS7_GrCtrlDB.InFault[297];
	      U   #Gr.OutWarning;
	      =   GCS7_GrCtrlDB.InWarning[297];
	      U   #Gr.OutManual;
	      =   GCS7_GrCtrlDB.InManual[297];
	      U   #Gr.OutHWStop;
	      =   GCS7_GrCtrlDB.InHWStop[297];
	      U   #Gr.OutDPFault;
	      =   GCS7_GrCtrlDB.InDPFault[297];
	      U   #Gr.OutLoaded;
	      =   GCS7_GrCtrlDB.InLoaded[297];
	      U   #Gr.OutAutoStart;
	      =   GCS7_GrCtrlDB.InAutoStart[297];
	      U   #Gr.VarStartWarning;
	      =   GCS7_GrCtrlDB.InStartWarning[297];
	NETWORK
	TITLE =End of block

	BE

	END_FUNCTION_BLOCK
